// TIA Portal V19 export
TYPE "LAF_typeSpecialFunctions"
TITLE = LAF_typeSpecialFunctions
// Commands to set Special Functions
// stored: Access Published
   STRUCT
      stopEndOfCycle : Bool;   // Command to stop at the end of the cycle
      initalPosition : Bool;   // Command to move to initial position
      releaseEntry : Bool;   // Command to release entry to an area
      dryRun : Bool;   // Command to run without parts
      specialFunction05 : Bool;   // Command for user defined special function
      specialFunction06 : Bool;   // Command for user defined special function
      specialFunction07 : Bool;   // Command for user defined special function
      specialFunction08 : Bool;   // Command for user defined special function
      specialFunction09 : Bool;   // Command for user defined special function
      specialFunction10 : Bool;   // Command for user defined special function
      specialFunction11 : Bool;   // Command for user defined special function
      specialFunction12 : Bool;   // Command for user defined special function
      specialFunction13 : Bool;   // Command for user defined special function
      specialFunction14 : Bool;   // Command for user defined special function
      specialFunction15 : Bool;   // Command for user defined special function
      specialFunction16 : Bool;   // Command for user defined special function
   END_STRUCT;
END_TYPE
